TYPE "StatusArea"
VERSION : 0.1
// Block: StatusArea
   STRUCT
      WarningPresence : Bool;
      AlarmPresence : Bool;
      WarningsNumber : Int;
      AlarmsNumber : Int;
      Status : Int;
   END_STRUCT;

END_TYPE
